// TIA Portal V19 export
TYPE "SpeedMachine_Config"
// stored: Access Published
   STRUCT
      SLS_VEL : LReal;
      DelayMissingCondition { ExternalVisible := 'False'} : Time;
      Ax : Struct
         SINA_Drive : "SpeedMotor_Config";
         MinAccTime : LReal := 0.1;
         MinDecTime : LReal := 0.1;
         LeadScrewPitchVal : LReal;
         MotorRevolution : LReal;
         LoadRevolution : LReal;
         PowerOffDelay : Time;
         StandstillVelocity : LReal;
         StandstillDelay : Time;
      END_STRUCT;
      Fan : Struct
         Presence : Bool;
         DelayOff : Time;
      END_STRUCT;
      Brake_Presence : Bool;
   END_STRUCT;
END_TYPE
